TYPE "PPrf_CoilHandling_WeldingCycle"
VERSION : 0.1
// Block: PPrf_CoilHandling_WeldingCycle
   STRUCT
      MeasureSheetEdgeReference : LReal;
      CorrStartWelding : LReal;
      CorrStopWelding : LReal;
   END_STRUCT;

END_TYPE
